(* IEC 61131-3 sources: mect_apps/TPAC1007_03/Latency_PLC, 4 files *)

(* ---- Crosstable.gvl ---- *)
VAR_GLOBAL
RISING_FRONT AT %IX0.772.0:BOOL;
FALLING_FRONT AT %IX0.776.0:BOOL;
PLC_FWrevision AT %IW0.21200:UINT;
PLC_HWconfig AT %IW0.21204:UINT;
PLC_DigDir_1 AT %QX0.21208.0:BOOL;
PLC_DigDir_2 AT %QX0.21212.0:BOOL;
PLC_DigDir_3 AT %QX0.21216.0:BOOL;
PLC_DigDir_4 AT %QX0.21220.0:BOOL;
PLC_DigDir_5 AT %QX0.21224.0:BOOL;
PLC_DigDir_6 AT %QX0.21228.0:BOOL;
PLC_DigDir_7 AT %QX0.21232.0:BOOL;
PLC_DigDir_8 AT %QX0.21236.0:BOOL;
PLC_AnInConf_1 AT %QW0.21240:UINT;
PLC_AnInConf_2 AT %QW0.21244:UINT;
PLC_AnOutConf_1 AT %QW0.21248:UINT;
PLC_DigIn_1 AT %IX0.21252.0:BOOL;
PLC_DigIn_2 AT %IX0.21256.0:BOOL;
PLC_DigIn_3 AT %IX0.21260.0:BOOL;
PLC_DigIn_4 AT %IX0.21264.0:BOOL;
PLC_DigIn_5 AT %IX0.21268.0:BOOL;
PLC_DigIn_6 AT %IX0.21272.0:BOOL;
PLC_DigIn_7 AT %IX0.21276.0:BOOL;
PLC_DigIn_8 AT %IX0.21280.0:BOOL;
PLC_DigIn_9 AT %IX0.21284.0:BOOL;
PLC_DigIn_10 AT %IX0.21288.0:BOOL;
PLC_DigIn_11 AT %IX0.21292.0:BOOL;
PLC_DigIn_12 AT %IX0.21296.0:BOOL;
PLC_AnIn_1 AT %IW0.21300:INT;
PLC_AnIn_2 AT %IW0.21304:INT;
PLC_Tamb AT %IW0.21308:INT;
PLC_Encoder AT %ID0.21312:UDINT;
PLC_DigOut_1 AT %QX0.21316.0:BOOL;
PLC_DigOut_2 AT %QX0.21320.0:BOOL;
PLC_DigOut_3 AT %QX0.21324.0:BOOL;
PLC_DigOut_4 AT %QX0.21328.0:BOOL;
PLC_DigOut_5 AT %QX0.21332.0:BOOL;
PLC_DigOut_6 AT %QX0.21336.0:BOOL;
PLC_DigOut_7 AT %QX0.21340.0:BOOL;
PLC_DigOut_8 AT %QX0.21344.0:BOOL;
PLC_AnOut_1 AT %QW0.21348:INT;
PLC_EncEnable AT %QW0.21352:UINT;
PLC_EncoderReset AT %QW0.21356:UINT;
PLC_Reserved_16 AT %QW0.21360:UINT;
PLC_Reserved_17 AT %QW0.21364:UINT;
PLC_Reserved_18 AT %QW0.21368:UINT;
PLC_Reserved_19 AT %QW0.21372:UINT;
PLC_Heartbeat AT %IW0.21376:UINT;
PLC_time AT %ID0.21560:REAL;
PLC_timeMin AT %ID0.21564:REAL;
PLC_timeMax AT %ID0.21568:REAL;
PLC_timeWin AT %QD0.21572:REAL;
PLC_Version AT %IW0.21576:UINT;
PLC_EngineStatus AT %IW0.21580:UINT;
PLC_ResetValues AT %QX0.21584.0:BOOL;
END_VAR

(* ---- Events.st ---- *)
(*[[
]]*)
PROGRAM Events
#import "Crosstable.gvl"
VAR
END_VAR

	if RISING_FRONT then
		PLC_DigOut_6 := TRUE;
	end_if;
	if FALLING_FRONT then
		PLC_DigOut_6 := FALSE;
	end_if;

END_PROGRAM

(* ---- Init.st ---- *)
(*[[
]]*)
PROGRAM Init
#import "Crosstable.gvl"

	PLC_DigDir_5 := 0; (* Latency Input *)
	PLC_DigDir_6 := 1; (* Latency Output *)

	PLC_AnInConf_1 := 2; (* 0..10V *)
	PLC_AnInConf_2 := 2; (* 0..10V *)
	PLC_AnOutConf_1 := 2; (* 0..10V *)

END_PROGRAM

(* ---- Normal.st ---- *)
(*[[
]]*)
PROGRAM Normal
#import "Resource1.gvl"
#import "Crosstable.gvl"

VAR
	first : BOOL := TRUE;
	timer : TON;
	flip : BOOL := TRUE;
END_VAR;

	if first then
		first := false;

		(* digital i/o configuration *)
		PLC_DigDir_1 := 1; (* output *)
		PLC_DigDir_2 := 1; (* output *)
		PLC_DigDir_3 := 1; (* output *)
		PLC_DigDir_4 := 1; (* output *)
		PLC_DigDir_5 := 0; (* input *)
		PLC_DigDir_6 := 0; (* input *)
		PLC_DigDir_7 := 1; (* output *)
		PLC_DigDir_8 := 0; (* input *)

		(* analog i/o configuration *)
		PLC_AnInConf_1 := 2; (* voltage *)
		PLC_AnInConf_2 := 2; (* voltage *)
		PLC_AnOutConf_1 := 2; (* voltage *)
	end_if;

	(* work load *)
	timer(IN := TRUE, PT := T#500ms );
	if timer.Q then
		flip := not flip;
		PLC_DigOut_7 := flip;
		PLC_AnOut_1 := ((PLC_AnIn_1 + PLC_AnIn_2) / 2) / 10;
		timer(IN := FALSE);
		timer(IN := TRUE);
	end_if;

END_PROGRAM
